(* Logix 5000 project; controller LeakTestAuto vendor 1 type 14 code 226 rev 37.11; software revision 37.01; part 4 of 13 *)

        [2].Detailed.element_data[13].result_measurement := 0.00085681677, [2].Detailed.element_data[14].Variable_code := 218, [2].Detailed.element_data[14].prec_code := 3, [2].Detailed.element_data[14].Unit_code := 41, [2].Detailed.element_data[14].result_measurement := 0.01094304, [2].Detailed.element_data[15].Variable_code := 295, [2].Detailed.element_data[15].prec_code := 3, [2].Detailed.element_data[15].Unit_code := 12, [2].Detailed.element_data[15].result_measurement := 5.073389, [3].UID := 10574, [3].Basic.unique_id := 10574, [3].Basic.channel_num := 1, [3].Basic.program_num := 2, [3].Basic.evaluation_code := 1, [3].Basic.test_port := 1, [3].Basic.year := 26, [3].Basic.month := 9, [3].Basic.date := 25, [3].Basic.hour := 12, [3].Basic.minute := 22, [3].Basic.second := 21, [3].Basic.flags := 12, [3].Basic.Num_tests := 1, [3].Basic.test_elements.test_type := 66, [3].Basic.test_elements.test_eval := 1, [3].Basic.test_elements.num_elements := 16, [3].Detailed.unique_id := 10574, [3].Detailed.num_elements := 16, [3].Detailed.Test_Type := 66, [3].Detailed.element_data[0].Variable_code := 61, [3].Detailed.element_data[0].prec_code := 2, [3].Detailed.element_data[0].Unit_code := 60, [3].Detailed.element_data[0].result_measurement := 0.11958182, [3].Detailed.element_data[1].Variable_code := 28, [3].Detailed.element_data[1].prec_code := 3, [3].Detailed.element_data[1].Unit_code := 41, [3].Detailed.element_data[1].result_measurement := 0.0037439167, [3].Detailed.element_data[2].Variable_code := 13, [3].Detailed.element_data[2].prec_code := 3, [3].Detailed.element_data[2].Unit_code := 12, [3].Detailed.element_data[2].result_measurement := 5.0675263, [3].Detailed.element_data[3].Variable_code := 75, [3].Detailed.element_data[3].prec_code := 2, [3].Detailed.element_data[3].Unit_code := 60, [3].Detailed.element_data[4].Variable_code := 60, [3].Detailed.element_data[4].prec_code := 2, [3].Detailed.element_data[4].Unit_code := 60, [3].Detailed.element_data[4].result_measurement := 0.1301989, [3].Detailed.element_data[5].Variable_code := 56, [3].Detailed.element_data[5].prec_code := 3, [3].Detailed.element_data[5].Unit_code := 41, [3].Detailed.element_data[5].result_measurement := 0.0020628795, [3].Detailed.element_data[6].Variable_code := 55, [3].Detailed.element_data[6].prec_code := 3, [3].Detailed.element_data[6].Unit_code := 12, [3].Detailed.element_data[6].result_measurement := 5.0675263, [3].Detailed.element_data[7].Variable_code := 58, [3].Detailed.element_data[7].prec_code := 2, [3].Detailed.element_data[7].Unit_code := 60, [3].Detailed.element_data[7].result_measurement := -1.0002404,
        [3].Detailed.element_data[8].Variable_code := 59, [3].Detailed.element_data[8].prec_code := 2, [3].Detailed.element_data[8].Unit_code := 60, [3].Detailed.element_data[8].result_measurement := 1.0002404, [3].Detailed.element_data[9].Variable_code := 12, [3].Detailed.element_data[9].prec_code := 3, [3].Detailed.element_data[9].Unit_code := 12, [3].Detailed.element_data[9].result_measurement := 5.000001, [3].Detailed.element_data[10].Variable_code := 62, [3].Detailed.element_data[10].prec_code := 2, [3].Detailed.element_data[10].Unit_code := 60, [3].Detailed.element_data[10].result_measurement := 1.0902061, [3].Detailed.element_data[11].Variable_code := 21, [3].Detailed.element_data[11].prec_code := 3, [3].Detailed.element_data[11].Unit_code := 41, [3].Detailed.element_data[11].result_measurement := 0.0015180558, [3].Detailed.element_data[12].Variable_code := 25, [3].Detailed.element_data[12].prec_code := 3, [3].Detailed.element_data[12].Unit_code := 41, [3].Detailed.element_data[12].result_measurement := 0.021727756, [3].Detailed.element_data[13].Variable_code := 216, [3].Detailed.element_data[13].prec_code := 3, [3].Detailed.element_data[13].Unit_code := 41, [3].Detailed.element_data[13].result_measurement := 0.00085681677, [3].Detailed.element_data[14].Variable_code := 218, [3].Detailed.element_data[14].prec_code := 3, [3].Detailed.element_data[14].Unit_code := 41, [3].Detailed.element_data[14].result_measurement := 0.01094304, [3].Detailed.element_data[15].Variable_code := 295, [3].Detailed.element_data[15].prec_code := 3, [3].Detailed.element_data[15].Unit_code := 12, [3].Detailed.element_data[15].result_measurement := 5.0734262, [4].UID := 10577, [4].Basic.unique_id := 10577, [4].Basic.channel_num := 1, [4].Basic.program_num := 2, [4].Basic.evaluation_code := 1, [4].Basic.test_port := 1, [4].Basic.year := 26, [4].Basic.month := 9, [4].Basic.date := 25, [4].Basic.hour := 12, [4].Basic.minute := 22, [4].Basic.second := 54, [4].Basic.flags := 12, [4].Basic.Num_tests := 1, [4].Basic.test_elements.test_type := 66, [4].Basic.test_elements.test_eval := 1, [4].Basic.test_elements.num_elements := 16, [4].Detailed.unique_id := 10577, [4].Detailed.num_elements := 16, [4].Detailed.Test_Type := 66, [4].Detailed.element_data[0].Variable_code := 61, [4].Detailed.element_data[0].prec_code := 2, [4].Detailed.element_data[0].Unit_code := 60, [4].Detailed.element_data[0].result_measurement := 0.10728836, [4].Detailed.element_data[1].Variable_code := 28, [4].Detailed.element_data[1].prec_code := 3, [4].Detailed.element_data[1].Unit_code := 41, [4].Detailed.element_data[1].result_measurement := 0.0035157427,
        [4].Detailed.element_data[2].Variable_code := 13, [4].Detailed.element_data[2].prec_code := 3, [4].Detailed.element_data[2].Unit_code := 12, [4].Detailed.element_data[2].result_measurement := 5.0673585, [4].Detailed.element_data[3].Variable_code := 75, [4].Detailed.element_data[3].prec_code := 2, [4].Detailed.element_data[3].Unit_code := 60, [4].Detailed.element_data[4].Variable_code := 60, [4].Detailed.element_data[4].prec_code := 2, [4].Detailed.element_data[4].Unit_code := 60, [4].Detailed.element_data[4].result_measurement := 0.093877316, [4].Detailed.element_data[5].Variable_code := 56, [4].Detailed.element_data[5].prec_code := 3, [4].Detailed.element_data[5].Unit_code := 41, [4].Detailed.element_data[5].result_measurement := 0.0017276034, [4].Detailed.element_data[6].Variable_code := 55, [4].Detailed.element_data[6].prec_code := 3, [4].Detailed.element_data[6].Unit_code := 12, [4].Detailed.element_data[6].result_measurement := 5.0673585, [4].Detailed.element_data[7].Variable_code := 58, [4].Detailed.element_data[7].prec_code := 2, [4].Detailed.element_data[7].Unit_code := 60, [4].Detailed.element_data[7].result_measurement := -1.0002404, [4].Detailed.element_data[8].Variable_code := 59, [4].Detailed.element_data[8].prec_code := 2, [4].Detailed.element_data[8].Unit_code := 60, [4].Detailed.element_data[8].result_measurement := 1.0002404, [4].Detailed.element_data[9].Variable_code := 12, [4].Detailed.element_data[9].prec_code := 3, [4].Detailed.element_data[9].Unit_code := 12, [4].Detailed.element_data[9].result_measurement := 5.000001, [4].Detailed.element_data[10].Variable_code := 62, [4].Detailed.element_data[10].prec_code := 2, [4].Detailed.element_data[10].Unit_code := 60, [4].Detailed.element_data[10].result_measurement := 1.0902061, [4].Detailed.element_data[11].Variable_code := 21, [4].Detailed.element_data[11].prec_code := 3, [4].Detailed.element_data[11].Unit_code := 41, [4].Detailed.element_data[11].result_measurement := 0.0015180558, [4].Detailed.element_data[12].Variable_code := 25, [4].Detailed.element_data[12].prec_code := 3, [4].Detailed.element_data[12].Unit_code := 41, [4].Detailed.element_data[12].result_measurement := 0.021727756, [4].Detailed.element_data[13].Variable_code := 216, [4].Detailed.element_data[13].prec_code := 3, [4].Detailed.element_data[13].Unit_code := 41, [4].Detailed.element_data[13].result_measurement := 0.00085681677, [4].Detailed.element_data[14].Variable_code := 218, [4].Detailed.element_data[14].prec_code := 3, [4].Detailed.element_data[14].Unit_code := 41, [4].Detailed.element_data[14].result_measurement := 0.01094304, [4].Detailed.element_data[15].Variable_code := 295, [4].Detailed.element_data[15].prec_code := 3, [4].Detailed.element_data[15].Unit_code := 12, [4].Detailed.element_data[15].result_measurement := 5.073468, [5].UID := 10580, [5].Basic.unique_id := 10580, [5].Basic.channel_num := 1, [5].Basic.program_num := 2, [5].Basic.evaluation_code := 1,
        [5].Basic.test_port := 1, [5].Basic.year := 26, [5].Basic.month := 9, [5].Basic.date := 25, [5].Basic.hour := 12, [5].Basic.minute := 27, [5].Basic.second := 36, [5].Basic.flags := 12, [5].Basic.Num_tests := 1, [5].Basic.test_elements.test_type := 66, [5].Basic.test_elements.test_eval := 1, [5].Basic.test_elements.num_elements := 16, [5].Detailed.unique_id := 10580, [5].Detailed.num_elements := 16, [5].Detailed.Test_Type := 66, [5].Detailed.element_data[0].Variable_code := 61, [5].Detailed.element_data[0].prec_code := 2, [5].Detailed.element_data[0].Unit_code := 60, [5].Detailed.element_data[0].result_measurement := 0.10281801, [5].Detailed.element_data[1].Variable_code := 28, [5].Detailed.element_data[1].prec_code := 3, [5].Detailed.element_data[1].Unit_code := 41, [5].Detailed.element_data[1].result_measurement := 0.003427267, [5].Detailed.element_data[2].Variable_code := 13, [5].Detailed.element_data[2].prec_code := 3, [5].Detailed.element_data[2].Unit_code := 12, [5].Detailed.element_data[2].result_measurement := 5.064076, [5].Detailed.element_data[3].Variable_code := 75, [5].Detailed.element_data[3].prec_code := 2, [5].Detailed.element_data[3].Unit_code := 60, [5].Detailed.element_data[4].Variable_code := 60, [5].Detailed.element_data[4].prec_code := 2, [5].Detailed.element_data[4].Unit_code := 60, [5].Detailed.element_data[4].result_measurement := 0.08773059, [5].Detailed.element_data[5].Variable_code := 56, [5].Detailed.element_data[5].prec_code := 3, [5].Detailed.element_data[5].Unit_code := 41, [5].Detailed.element_data[5].result_measurement := 0.001671724, [5].Detailed.element_data[6].Variable_code := 55, [5].Detailed.element_data[6].prec_code := 3, [5].Detailed.element_data[6].Unit_code := 12, [5].Detailed.element_data[6].result_measurement := 5.064076, [5].Detailed.element_data[7].Variable_code := 58, [5].Detailed.element_data[7].prec_code := 2, [5].Detailed.element_data[7].Unit_code := 60, [5].Detailed.element_data[7].result_measurement := -1.0002404, [5].Detailed.element_data[8].Variable_code := 59, [5].Detailed.element_data[8].prec_code := 2, [5].Detailed.element_data[8].Unit_code := 60, [5].Detailed.element_data[8].result_measurement := 1.0002404, [5].Detailed.element_data[9].Variable_code := 12, [5].Detailed.element_data[9].prec_code := 3, [5].Detailed.element_data[9].Unit_code := 12, [5].Detailed.element_data[9].result_measurement := 5.000001, [5].Detailed.element_data[10].Variable_code := 62, [5].Detailed.element_data[10].prec_code := 2, [5].Detailed.element_data[10].Unit_code := 60, [5].Detailed.element_data[10].result_measurement := 1.0902061, [5].Detailed.element_data[11].Variable_code := 21, [5].Detailed.element_data[11].prec_code := 3,
        [5].Detailed.element_data[11].Unit_code := 41, [5].Detailed.element_data[11].result_measurement := 0.0015180558, [5].Detailed.element_data[12].Variable_code := 25, [5].Detailed.element_data[12].prec_code := 3, [5].Detailed.element_data[12].Unit_code := 41, [5].Detailed.element_data[12].result_measurement := 0.021727756, [5].Detailed.element_data[13].Variable_code := 216, [5].Detailed.element_data[13].prec_code := 3, [5].Detailed.element_data[13].Unit_code := 41, [5].Detailed.element_data[13].result_measurement := 0.00085681677, [5].Detailed.element_data[14].Variable_code := 218, [5].Detailed.element_data[14].prec_code := 3, [5].Detailed.element_data[14].Unit_code := 41, [5].Detailed.element_data[14].result_measurement := 0.01094304, [5].Detailed.element_data[15].Variable_code := 295, [5].Detailed.element_data[15].prec_code := 3, [5].Detailed.element_data[15].Unit_code := 12, [5].Detailed.element_data[15].result_measurement := 5.0706367, [6].UID := 10583, [6].Basic.unique_id := 10583, [6].Basic.channel_num := 1, [6].Basic.program_num := 2, [6].Basic.evaluation_code := 1, [6].Basic.test_port := 1, [6].Basic.year := 26, [6].Basic.month := 9, [6].Basic.date := 25, [6].Basic.hour := 12, [6].Basic.minute := 28, [6].Basic.second := 6, [6].Basic.flags := 12, [6].Basic.Num_tests := 1, [6].Basic.test_elements.test_type := 66, [6].Basic.test_elements.test_eval := 1, [6].Basic.test_elements.num_elements := 16, [6].Detailed.unique_id := 10583, [6].Detailed.num_elements := 16, [6].Detailed.Test_Type := 66, [6].Detailed.element_data[0].Variable_code := 61, [6].Detailed.element_data[0].prec_code := 2, [6].Detailed.element_data[0].Unit_code := 60, [6].Detailed.element_data[0].result_measurement := 0.11622906, [6].Detailed.element_data[1].Variable_code := 28, [6].Detailed.element_data[1].prec_code := 3, [6].Detailed.element_data[1].Unit_code := 41, [6].Detailed.element_data[1].result_measurement := 0.0036740676, [6].Detailed.element_data[2].Variable_code := 13, [6].Detailed.element_data[2].prec_code := 3, [6].Detailed.element_data[2].Unit_code := 12, [6].Detailed.element_data[2].result_measurement := 5.0649743, [6].Detailed.element_data[3].Variable_code := 75, [6].Detailed.element_data[3].prec_code := 2, [6].Detailed.element_data[3].Unit_code := 60, [6].Detailed.element_data[4].Variable_code := 60, [6].Detailed.element_data[4].prec_code := 2, [6].Detailed.element_data[4].Unit_code := 60, [6].Detailed.element_data[4].result_measurement := 0.10114163, [6].Detailed.element_data[5].Variable_code := 56, [6].Detailed.element_data[5].prec_code := 3, [6].Detailed.element_data[5].Unit_code := 41,
        [6].Detailed.element_data[5].result_measurement := 0.001792796, [6].Detailed.element_data[6].Variable_code := 55, [6].Detailed.element_data[6].prec_code := 3, [6].Detailed.element_data[6].Unit_code := 12, [6].Detailed.element_data[6].result_measurement := 5.0649743, [6].Detailed.element_data[7].Variable_code := 58, [6].Detailed.element_data[7].prec_code := 2, [6].Detailed.element_data[7].Unit_code := 60, [6].Detailed.element_data[7].result_measurement := -1.0002404, [6].Detailed.element_data[8].Variable_code := 59, [6].Detailed.element_data[8].prec_code := 2, [6].Detailed.element_data[8].Unit_code := 60, [6].Detailed.element_data[8].result_measurement := 1.0002404, [6].Detailed.element_data[9].Variable_code := 12, [6].Detailed.element_data[9].prec_code := 3, [6].Detailed.element_data[9].Unit_code := 12, [6].Detailed.element_data[9].result_measurement := 5.000001, [6].Detailed.element_data[10].Variable_code := 62, [6].Detailed.element_data[10].prec_code := 2, [6].Detailed.element_data[10].Unit_code := 60, [6].Detailed.element_data[10].result_measurement := 1.0902061, [6].Detailed.element_data[11].Variable_code := 21, [6].Detailed.element_data[11].prec_code := 3, [6].Detailed.element_data[11].Unit_code := 41, [6].Detailed.element_data[11].result_measurement := 0.0015180558, [6].Detailed.element_data[12].Variable_code := 25, [6].Detailed.element_data[12].prec_code := 3, [6].Detailed.element_data[12].Unit_code := 41, [6].Detailed.element_data[12].result_measurement := 0.021727756, [6].Detailed.element_data[13].Variable_code := 216, [6].Detailed.element_data[13].prec_code := 3, [6].Detailed.element_data[13].Unit_code := 41, [6].Detailed.element_data[13].result_measurement := 0.00085681677, [6].Detailed.element_data[14].Variable_code := 218, [6].Detailed.element_data[14].prec_code := 3, [6].Detailed.element_data[14].Unit_code := 41, [6].Detailed.element_data[14].result_measurement := 0.01094304, [6].Detailed.element_data[15].Variable_code := 295, [6].Detailed.element_data[15].prec_code := 3, [6].Detailed.element_data[15].Unit_code := 12, [6].Detailed.element_data[15].result_measurement := 5.0712004, [7].UID := 10586, [7].Basic.unique_id := 10586, [7].Basic.channel_num := 1, [7].Basic.program_num := 2, [7].Basic.evaluation_code := 1, [7].Basic.test_port := 1, [7].Basic.year := 26, [7].Basic.month := 9, [7].Basic.date := 25, [7].Basic.hour := 12, [7].Basic.minute := 38, [7].Basic.second := 12, [7].Basic.flags := 12, [7].Basic.Num_tests := 1, [7].Basic.test_elements.test_type := 66, [7].Basic.test_elements.test_eval := 1, [7].Basic.test_elements.num_elements := 16, [7].Detailed.unique_id := 10586, [7].Detailed.num_elements := 16,
        [7].Detailed.Test_Type := 66, [7].Detailed.element_data[0].Variable_code := 61, [7].Detailed.element_data[0].prec_code := 2, [7].Detailed.element_data[0].Unit_code := 60, [7].Detailed.element_data[0].result_measurement := 0.11678785, [7].Detailed.element_data[1].Variable_code := 28, [7].Detailed.element_data[1].prec_code := 3, [7].Detailed.element_data[1].Unit_code := 41, [7].Detailed.element_data[1].result_measurement := 0.0036833808, [7].Detailed.element_data[2].Variable_code := 13, [7].Detailed.element_data[2].prec_code := 3, [7].Detailed.element_data[2].Unit_code := 12, [7].Detailed.element_data[2].result_measurement := 5.063303, [7].Detailed.element_data[3].Variable_code := 75, [7].Detailed.element_data[3].prec_code := 2, [7].Detailed.element_data[3].Unit_code := 60, [7].Detailed.element_data[4].Variable_code := 60, [7].Detailed.element_data[4].prec_code := 2, [7].Detailed.element_data[4].Unit_code := 60, [7].Detailed.element_data[4].result_measurement := 0.10617077, [7].Detailed.element_data[5].Variable_code := 56, [7].Detailed.element_data[5].prec_code := 3, [7].Detailed.element_data[5].Unit_code := 41, [7].Detailed.element_data[5].result_measurement := 0.0018440187, [7].Detailed.element_data[6].Variable_code := 55, [7].Detailed.element_data[6].prec_code := 3, [7].Detailed.element_data[6].Unit_code := 12, [7].Detailed.element_data[6].result_measurement := 5.063303, [7].Detailed.element_data[7].Variable_code := 58, [7].Detailed.element_data[7].prec_code := 2, [7].Detailed.element_data[7].Unit_code := 60, [7].Detailed.element_data[7].result_measurement := -1.0002404, [7].Detailed.element_data[8].Variable_code := 59, [7].Detailed.element_data[8].prec_code := 2, [7].Detailed.element_data[8].Unit_code := 60, [7].Detailed.element_data[8].result_measurement := 1.0002404, [7].Detailed.element_data[9].Variable_code := 12, [7].Detailed.element_data[9].prec_code := 3, [7].Detailed.element_data[9].Unit_code := 12, [7].Detailed.element_data[9].result_measurement := 5.000001, [7].Detailed.element_data[10].Variable_code := 62, [7].Detailed.element_data[10].prec_code := 2, [7].Detailed.element_data[10].Unit_code := 60, [7].Detailed.element_data[10].result_measurement := 1.0902061, [7].Detailed.element_data[11].Variable_code := 21, [7].Detailed.element_data[11].prec_code := 3, [7].Detailed.element_data[11].Unit_code := 41, [7].Detailed.element_data[11].result_measurement := 0.0015180558, [7].Detailed.element_data[12].Variable_code := 25, [7].Detailed.element_data[12].prec_code := 3, [7].Detailed.element_data[12].Unit_code := 41, [7].Detailed.element_data[12].result_measurement := 0.021727756, [7].Detailed.element_data[13].Variable_code := 216, [7].Detailed.element_data[13].prec_code := 3, [7].Detailed.element_data[13].Unit_code := 41, [7].Detailed.element_data[13].result_measurement := 0.00085681677, [7].Detailed.element_data[14].Variable_code := 218, [7].Detailed.element_data[14].prec_code := 3, [7].Detailed.element_data[14].Unit_code := 41, [7].Detailed.element_data[14].result_measurement := 0.01094304,
        [7].Detailed.element_data[15].Variable_code := 295, [7].Detailed.element_data[15].prec_code := 3, [7].Detailed.element_data[15].Unit_code := 12, [7].Detailed.element_data[15].result_measurement := 5.0700407, [8].UID := 10589, [8].Basic.unique_id := 10589, [8].Basic.channel_num := 1, [8].Basic.program_num := 2, [8].Basic.evaluation_code := 1, [8].Basic.test_port := 1, [8].Basic.year := 26, [8].Basic.month := 9, [8].Basic.date := 25, [8].Basic.hour := 12, [8].Basic.minute := 39, [8].Basic.second := 1, [8].Basic.flags := 12, [8].Basic.Num_tests := 1, [8].Basic.test_elements.test_type := 66, [8].Basic.test_elements.test_eval := 1, [8].Basic.test_elements.num_elements := 16, [8].Detailed.unique_id := 10589, [8].Detailed.num_elements := 16, [8].Detailed.Test_Type := 66, [8].Detailed.element_data[0].Variable_code := 61, [8].Detailed.element_data[0].prec_code := 2, [8].Detailed.element_data[0].Unit_code := 60, [8].Detailed.element_data[0].result_measurement := 0.11175871, [8].Detailed.element_data[1].Variable_code := 28, [8].Detailed.element_data[1].prec_code := 3, [8].Detailed.element_data[1].Unit_code := 41, [8].Detailed.element_data[1].result_measurement := 0.0035949051, [8].Detailed.element_data[2].Variable_code := 13, [8].Detailed.element_data[2].prec_code := 3, [8].Detailed.element_data[2].Unit_code := 12, [8].Detailed.element_data[2].result_measurement := 5.0623946, [8].Detailed.element_data[3].Variable_code := 75, [8].Detailed.element_data[3].prec_code := 2, [8].Detailed.element_data[3].Unit_code := 60, [8].Detailed.element_data[4].Variable_code := 60, [8].Detailed.element_data[4].prec_code := 2, [8].Detailed.element_data[4].Unit_code := 60, [8].Detailed.element_data[4].result_measurement := 0.11175871, [8].Detailed.element_data[5].Variable_code := 56, [8].Detailed.element_data[5].prec_code := 3, [8].Detailed.element_data[5].Unit_code := 41, [8].Detailed.element_data[5].result_measurement := 0.0018952414, [8].Detailed.element_data[6].Variable_code := 55, [8].Detailed.element_data[6].prec_code := 3, [8].Detailed.element_data[6].Unit_code := 12, [8].Detailed.element_data[6].result_measurement := 5.0623946, [8].Detailed.element_data[7].Variable_code := 58, [8].Detailed.element_data[7].prec_code := 2, [8].Detailed.element_data[7].Unit_code := 60, [8].Detailed.element_data[7].result_measurement := -1.0002404, [8].Detailed.element_data[8].Variable_code := 59, [8].Detailed.element_data[8].prec_code := 2, [8].Detailed.element_data[8].Unit_code := 60, [8].Detailed.element_data[8].result_measurement := 1.0002404, [8].Detailed.element_data[9].Variable_code := 12,
        [8].Detailed.element_data[9].prec_code := 3, [8].Detailed.element_data[9].Unit_code := 12, [8].Detailed.element_data[9].result_measurement := 5.000001, [8].Detailed.element_data[10].Variable_code := 62, [8].Detailed.element_data[10].prec_code := 2, [8].Detailed.element_data[10].Unit_code := 60, [8].Detailed.element_data[10].result_measurement := 1.0902061, [8].Detailed.element_data[11].Variable_code := 21, [8].Detailed.element_data[11].prec_code := 3, [8].Detailed.element_data[11].Unit_code := 41, [8].Detailed.element_data[11].result_measurement := 0.0015180558, [8].Detailed.element_data[12].Variable_code := 25, [8].Detailed.element_data[12].prec_code := 3, [8].Detailed.element_data[12].Unit_code := 41, [8].Detailed.element_data[12].result_measurement := 0.021727756, [8].Detailed.element_data[13].Variable_code := 216, [8].Detailed.element_data[13].prec_code := 3, [8].Detailed.element_data[13].Unit_code := 41, [8].Detailed.element_data[13].result_measurement := 0.00085681677, [8].Detailed.element_data[14].Variable_code := 218, [8].Detailed.element_data[14].prec_code := 3, [8].Detailed.element_data[14].Unit_code := 41, [8].Detailed.element_data[14].result_measurement := 0.01094304, [8].Detailed.element_data[15].Variable_code := 295, [8].Detailed.element_data[15].prec_code := 3, [8].Detailed.element_data[15].Unit_code := 12, [8].Detailed.element_data[15].result_measurement := 5.068914, [9].UID := 10592, [9].Basic.unique_id := 10592, [9].Basic.channel_num := 1, [9].Basic.program_num := 2, [9].Basic.evaluation_code := 1, [9].Basic.test_port := 1, [9].Basic.year := 26, [9].Basic.month := 9, [9].Basic.date := 25, [9].Basic.hour := 12, [9].Basic.minute := 39, [9].Basic.second := 32, [9].Basic.flags := 12, [9].Basic.Num_tests := 1, [9].Basic.test_elements.test_type := 66, [9].Basic.test_elements.test_eval := 1, [9].Basic.test_elements.num_elements := 16, [9].Detailed.unique_id := 10592, [9].Detailed.num_elements := 16, [9].Detailed.Test_Type := 66, [9].Detailed.element_data[0].Variable_code := 61, [9].Detailed.element_data[0].prec_code := 2, [9].Detailed.element_data[0].Unit_code := 60, [9].Detailed.element_data[0].result_measurement := 0.10728836, [9].Detailed.element_data[1].Variable_code := 28, [9].Detailed.element_data[1].prec_code := 3, [9].Detailed.element_data[1].Unit_code := 41, [9].Detailed.element_data[1].result_measurement := 0.003511086, [9].Detailed.element_data[2].Variable_code := 13, [9].Detailed.element_data[2].prec_code := 3, [9].Detailed.element_data[2].Unit_code := 12, [9].Detailed.element_data[2].result_measurement := 5.0658684, [9].Detailed.element_data[3].Variable_code := 75,
        [9].Detailed.element_data[3].prec_code := 2, [9].Detailed.element_data[3].Unit_code := 60, [9].Detailed.element_data[4].Variable_code := 60, [9].Detailed.element_data[4].prec_code := 2, [9].Detailed.element_data[4].Unit_code := 60, [9].Detailed.element_data[4].result_measurement := 0.12684613, [9].Detailed.element_data[5].Variable_code := 56, [9].Detailed.element_data[5].prec_code := 3, [9].Detailed.element_data[5].Unit_code := 41, [9].Detailed.element_data[5].result_measurement := 0.0020349398, [9].Detailed.element_data[6].Variable_code := 55, [9].Detailed.element_data[6].prec_code := 3, [9].Detailed.element_data[6].Unit_code := 12, [9].Detailed.element_data[6].result_measurement := 5.0658684, [9].Detailed.element_data[7].Variable_code := 58, [9].Detailed.element_data[7].prec_code := 2, [9].Detailed.element_data[7].Unit_code := 60, [9].Detailed.element_data[7].result_measurement := -1.0002404, [9].Detailed.element_data[8].Variable_code := 59, [9].Detailed.element_data[8].prec_code := 2, [9].Detailed.element_data[8].Unit_code := 60, [9].Detailed.element_data[8].result_measurement := 1.0002404, [9].Detailed.element_data[9].Variable_code := 12, [9].Detailed.element_data[9].prec_code := 3, [9].Detailed.element_data[9].Unit_code := 12, [9].Detailed.element_data[9].result_measurement := 5.000001, [9].Detailed.element_data[10].Variable_code := 62, [9].Detailed.element_data[10].prec_code := 2, [9].Detailed.element_data[10].Unit_code := 60, [9].Detailed.element_data[10].result_measurement := 1.0902061, [9].Detailed.element_data[11].Variable_code := 21, [9].Detailed.element_data[11].prec_code := 3, [9].Detailed.element_data[11].Unit_code := 41, [9].Detailed.element_data[11].result_measurement := 0.0015180558, [9].Detailed.element_data[12].Variable_code := 25, [9].Detailed.element_data[12].prec_code := 3, [9].Detailed.element_data[12].Unit_code := 41, [9].Detailed.element_data[12].result_measurement := 0.021727756, [9].Detailed.element_data[13].Variable_code := 216, [9].Detailed.element_data[13].prec_code := 3, [9].Detailed.element_data[13].Unit_code := 41, [9].Detailed.element_data[13].result_measurement := 0.00085681677, [9].Detailed.element_data[14].Variable_code := 218, [9].Detailed.element_data[14].prec_code := 3, [9].Detailed.element_data[14].Unit_code := 41, [9].Detailed.element_data[14].result_measurement := 0.01094304, [9].Detailed.element_data[15].Variable_code := 295, [9].Detailed.element_data[15].prec_code := 3, [9].Detailed.element_data[15].Unit_code := 12, [9].Detailed.element_data[15].result_measurement := 5.0730352);
   CTS2_ResultHistoryVol : udt_CTS_RESULT[10] := ([0].UID := 10564, [0].Basic.unique_id := 10564, [0].Basic.channel_num := 1, [0].Basic.program_num := 1, [0].Basic.evaluation_code := 1, [0].Basic.test_port := 1, [0].Basic.year := 26, [0].Basic.month := 9, [0].Basic.date := 25, [0].Basic.hour := 12, [0].Basic.minute := 21, [0].Basic.second := 12, [0].Basic.flags := 12, [0].Basic.Num_tests := 1, [0].Basic.test_elements.test_type := 69, [0].Basic.test_elements.test_eval := 1, [0].Basic.test_elements.num_elements := 4, [0].Detailed.unique_id := 10564, [0].Detailed.num_elements := 4, [0].Detailed.Test_Type := 69, [0].Detailed.element_data[0].Variable_code := 245, [0].Detailed.element_data[0].prec_code := 2, [0].Detailed.element_data[0].Unit_code := 165, [0].Detailed.element_data[0].result_measurement := 156.89374, [0].Detailed.element_data[1].Variable_code := 13, [0].Detailed.element_data[1].prec_code := 3, [0].Detailed.element_data[1].Unit_code := 12, [0].Detailed.element_data[1].result_measurement := 1.962753, [0].Detailed.element_data[2].Variable_code := 247, [0].Detailed.element_data[2].prec_code := 3, [0].Detailed.element_data[2].Unit_code := 12, [0].Detailed.element_data[2].result_measurement := 5.0421896, [0].Detailed.element_data[3].Variable_code := 295, [0].Detailed.element_data[3].prec_code := 3, [0].Detailed.element_data[3].Unit_code := 12, [0].Detailed.element_data[3].result_measurement := 5.0442944, [1].UID := 10567, [1].Basic.unique_id := 10567, [1].Basic.channel_num := 1, [1].Basic.program_num := 1, [1].Basic.evaluation_code := 1, [1].Basic.test_port := 1, [1].Basic.year := 26, [1].Basic.month := 9, [1].Basic.date := 25, [1].Basic.hour := 12, [1].Basic.minute := 21, [1].Basic.second := 33, [1].Basic.flags := 12, [1].Basic.Num_tests := 1, [1].Basic.test_elements.test_type := 69, [1].Basic.test_elements.test_eval := 1, [1].Basic.test_elements.num_elements := 4, [1].Detailed.unique_id := 10567, [1].Detailed.num_elements := 4, [1].Detailed.Test_Type := 69, [1].Detailed.element_data[0].Variable_code := 245, [1].Detailed.element_data[0].prec_code := 2, [1].Detailed.element_data[0].Unit_code := 165, [1].Detailed.element_data[0].result_measurement := 156.82765,
        [1].Detailed.element_data[1].Variable_code := 13, [1].Detailed.element_data[1].prec_code := 3, [1].Detailed.element_data[1].Unit_code := 12, [1].Detailed.element_data[1].result_measurement := 1.9633397, [1].Detailed.element_data[2].Variable_code := 247, [1].Detailed.element_data[2].prec_code := 3, [1].Detailed.element_data[2].Unit_code := 12, [1].Detailed.element_data[2].result_measurement := 5.0423994, [1].Detailed.element_data[3].Variable_code := 295, [1].Detailed.element_data[3].prec_code := 3, [1].Detailed.element_data[3].Unit_code := 12, [1].Detailed.element_data[3].result_measurement := 5.04469, [2].UID := 10570, [2].Basic.unique_id := 10570, [2].Basic.channel_num := 1, [2].Basic.program_num := 1, [2].Basic.evaluation_code := 1, [2].Basic.test_port := 1, [2].Basic.year := 26, [2].Basic.month := 9, [2].Basic.date := 25, [2].Basic.hour := 12, [2].Basic.minute := 21, [2].Basic.second := 54, [2].Basic.flags := 12, [2].Basic.Num_tests := 1, [2].Basic.test_elements.test_type := 69, [2].Basic.test_elements.test_eval := 1, [2].Basic.test_elements.num_elements := 4, [2].Detailed.unique_id := 10570, [2].Detailed.num_elements := 4, [2].Detailed.Test_Type := 69, [2].Detailed.element_data[0].Variable_code := 245, [2].Detailed.element_data[0].prec_code := 2, [2].Detailed.element_data[0].Unit_code := 165, [2].Detailed.element_data[0].result_measurement := 156.6537, [2].Detailed.element_data[1].Variable_code := 13, [2].Detailed.element_data[1].prec_code := 3, [2].Detailed.element_data[1].Unit_code := 12, [2].Detailed.element_data[1].result_measurement := 1.9648718, [2].Detailed.element_data[2].Variable_code := 247, [2].Detailed.element_data[2].prec_code := 3, [2].Detailed.element_data[2].Unit_code := 12, [2].Detailed.element_data[2].result_measurement := 5.0429163, [2].Detailed.element_data[3].Variable_code := 295, [2].Detailed.element_data[3].prec_code := 3, [2].Detailed.element_data[3].Unit_code := 12, [2].Detailed.element_data[3].result_measurement := 5.044765, [3].UID := 10573, [3].Basic.unique_id := 10573, [3].Basic.channel_num := 1, [3].Basic.program_num := 1, [3].Basic.evaluation_code := 1, [3].Basic.test_port := 1, [3].Basic.year := 26, [3].Basic.month := 9, [3].Basic.date := 25, [3].Basic.hour := 12, [3].Basic.minute := 22, [3].Basic.second := 15,
        [3].Basic.flags := 12, [3].Basic.Num_tests := 1, [3].Basic.test_elements.test_type := 69, [3].Basic.test_elements.test_eval := 1, [3].Basic.test_elements.num_elements := 4, [3].Detailed.unique_id := 10573, [3].Detailed.num_elements := 4, [3].Detailed.Test_Type := 69, [3].Detailed.element_data[0].Variable_code := 245, [3].Detailed.element_data[0].prec_code := 2, [3].Detailed.element_data[0].Unit_code := 165, [3].Detailed.element_data[0].result_measurement := 156.76877, [3].Detailed.element_data[1].Variable_code := 13, [3].Detailed.element_data[1].prec_code := 3, [3].Detailed.element_data[1].Unit_code := 12, [3].Detailed.element_data[1].result_measurement := 1.9644899, [3].Detailed.element_data[2].Variable_code := 247, [3].Detailed.element_data[2].prec_code := 3, [3].Detailed.element_data[2].Unit_code := 12, [3].Detailed.element_data[2].result_measurement := 5.0441966, [3].Detailed.element_data[3].Variable_code := 295, [3].Detailed.element_data[3].prec_code := 3, [3].Detailed.element_data[3].Unit_code := 12, [3].Detailed.element_data[3].result_measurement := 5.0450954, [4].UID := 10576, [4].Basic.unique_id := 10576, [4].Basic.channel_num := 1, [4].Basic.program_num := 1, [4].Basic.evaluation_code := 1, [4].Basic.test_port := 1, [4].Basic.year := 26, [4].Basic.month := 9, [4].Basic.date := 25, [4].Basic.hour := 12, [4].Basic.minute := 22, [4].Basic.second := 47, [4].Basic.flags := 12, [4].Basic.Num_tests := 1, [4].Basic.test_elements.test_type := 69, [4].Basic.test_elements.test_eval := 1, [4].Basic.test_elements.num_elements := 4, [4].Detailed.unique_id := 10576, [4].Detailed.num_elements := 4, [4].Detailed.Test_Type := 69, [4].Detailed.element_data[0].Variable_code := 245, [4].Detailed.element_data[0].prec_code := 2, [4].Detailed.element_data[0].Unit_code := 165, [4].Detailed.element_data[0].result_measurement := 154.13881, [4].Detailed.element_data[1].Variable_code := 13, [4].Detailed.element_data[1].prec_code := 3, [4].Detailed.element_data[1].Unit_code := 12, [4].Detailed.element_data[1].result_measurement := 1.9848579, [4].Detailed.element_data[2].Variable_code := 247, [4].Detailed.element_data[2].prec_code := 3, [4].Detailed.element_data[2].Unit_code := 12, [4].Detailed.element_data[2].result_measurement := 5.0442944, [4].Detailed.element_data[3].Variable_code := 295, [4].Detailed.element_data[3].prec_code := 3, [4].Detailed.element_data[3].Unit_code := 12, [4].Detailed.element_data[3].result_measurement := 5.0455236,
        [5].UID := 10579, [5].Basic.unique_id := 10579, [5].Basic.channel_num := 1, [5].Basic.program_num := 1, [5].Basic.evaluation_code := 1, [5].Basic.test_port := 1, [5].Basic.year := 26, [5].Basic.month := 9, [5].Basic.date := 25, [5].Basic.hour := 12, [5].Basic.minute := 27, [5].Basic.second := 29, [5].Basic.flags := 12, [5].Basic.Num_tests := 1, [5].Basic.test_elements.test_type := 69, [5].Basic.test_elements.test_eval := 1, [5].Basic.test_elements.num_elements := 4, [5].Detailed.unique_id := 10579, [5].Detailed.num_elements := 4, [5].Detailed.Test_Type := 69, [5].Detailed.element_data[0].Variable_code := 245, [5].Detailed.element_data[0].prec_code := 2, [5].Detailed.element_data[0].Unit_code := 165, [5].Detailed.element_data[0].result_measurement := 157.14537, [5].Detailed.element_data[1].Variable_code := 13, [5].Detailed.element_data[1].prec_code := 3, [5].Detailed.element_data[1].Unit_code := 12, [5].Detailed.element_data[1].result_measurement := 1.9622269, [5].Detailed.element_data[2].Variable_code := 247, [5].Detailed.element_data[2].prec_code := 3, [5].Detailed.element_data[2].Unit_code := 12, [5].Detailed.element_data[2].result_measurement := 5.0457754, [5].Detailed.element_data[3].Variable_code := 295, [5].Detailed.element_data[3].prec_code := 3, [5].Detailed.element_data[3].Unit_code := 12, [5].Detailed.element_data[3].result_measurement := 5.0467906, [6].UID := 10582, [6].Basic.unique_id := 10582, [6].Basic.channel_num := 1, [6].Basic.program_num := 1, [6].Basic.evaluation_code := 1, [6].Basic.test_port := 1, [6].Basic.year := 26, [6].Basic.month := 9, [6].Basic.date := 25, [6].Basic.hour := 12, [6].Basic.minute := 28, [6].Basic.flags := 12, [6].Basic.Num_tests := 1, [6].Basic.test_elements.test_type := 69, [6].Basic.test_elements.test_eval := 1, [6].Basic.test_elements.num_elements := 4, [6].Detailed.unique_id := 10582, [6].Detailed.num_elements := 4, [6].Detailed.Test_Type := 69, [6].Detailed.element_data[0].Variable_code := 245, [6].Detailed.element_data[0].prec_code := 2, [6].Detailed.element_data[0].Unit_code := 165, [6].Detailed.element_data[0].result_measurement := 156.1754, [6].Detailed.element_data[1].Variable_code := 13,
        [6].Detailed.element_data[1].prec_code := 3, [6].Detailed.element_data[1].Unit_code := 12, [6].Detailed.element_data[1].result_measurement := 1.9685458, [6].Detailed.element_data[2].Variable_code := 247, [6].Detailed.element_data[2].prec_code := 3, [6].Detailed.element_data[2].Unit_code := 12, [6].Detailed.element_data[2].result_measurement := 5.04293, [6].Detailed.element_data[3].Variable_code := 295, [6].Detailed.element_data[3].prec_code := 3, [6].Detailed.element_data[3].Unit_code := 12, [6].Detailed.element_data[3].result_measurement := 5.0441875, [7].UID := 10585, [7].Basic.unique_id := 10585, [7].Basic.channel_num := 1, [7].Basic.program_num := 1, [7].Basic.evaluation_code := 1, [7].Basic.test_port := 1, [7].Basic.year := 26, [7].Basic.month := 9, [7].Basic.date := 25, [7].Basic.hour := 12, [7].Basic.minute := 38, [7].Basic.second := 5, [7].Basic.flags := 12, [7].Basic.Num_tests := 1, [7].Basic.test_elements.test_type := 69, [7].Basic.test_elements.test_eval := 1, [7].Basic.test_elements.num_elements := 4, [7].Detailed.unique_id := 10585, [7].Detailed.num_elements := 4, [7].Detailed.Test_Type := 69, [7].Detailed.element_data[0].Variable_code := 245, [7].Detailed.element_data[0].prec_code := 2, [7].Detailed.element_data[0].Unit_code := 165, [7].Detailed.element_data[0].result_measurement := 156.68964, [7].Detailed.element_data[1].Variable_code := 13, [7].Detailed.element_data[1].prec_code := 3, [7].Detailed.element_data[1].Unit_code := 12, [7].Detailed.element_data[1].result_measurement := 1.9655237, [7].Detailed.element_data[2].Variable_code := 247, [7].Detailed.element_data[2].prec_code := 3, [7].Detailed.element_data[2].Unit_code := 12, [7].Detailed.element_data[2].result_measurement := 5.0452957, [7].Detailed.element_data[3].Variable_code := 295, [7].Detailed.element_data[3].prec_code := 3, [7].Detailed.element_data[3].Unit_code := 12, [7].Detailed.element_data[3].result_measurement := 5.046395, [8].UID := 10588, [8].Basic.unique_id := 10588, [8].Basic.channel_num := 1, [8].Basic.program_num := 1, [8].Basic.evaluation_code := 1, [8].Basic.test_port := 1, [8].Basic.year := 26, [8].Basic.month := 9, [8].Basic.date := 25, [8].Basic.hour := 12, [8].Basic.minute := 38, [8].Basic.second := 54, [8].Basic.flags := 12,
        [8].Basic.Num_tests := 1, [8].Basic.test_elements.test_type := 69, [8].Basic.test_elements.test_eval := 1, [8].Basic.test_elements.num_elements := 4, [8].Detailed.unique_id := 10588, [8].Detailed.num_elements := 4, [8].Detailed.Test_Type := 69, [8].Detailed.element_data[0].Variable_code := 245, [8].Detailed.element_data[0].prec_code := 2, [8].Detailed.element_data[0].Unit_code := 165, [8].Detailed.element_data[0].result_measurement := 156.9294, [8].Detailed.element_data[1].Variable_code := 13, [8].Detailed.element_data[1].prec_code := 3, [8].Detailed.element_data[1].Unit_code := 12, [8].Detailed.element_data[1].result_measurement := 1.9627343, [8].Detailed.element_data[2].Variable_code := 247, [8].Detailed.element_data[2].prec_code := 3, [8].Detailed.element_data[2].Unit_code := 12, [8].Detailed.element_data[2].result_measurement := 5.0428414, [8].Detailed.element_data[3].Variable_code := 295, [8].Detailed.element_data[3].prec_code := 3, [8].Detailed.element_data[3].Unit_code := 12, [8].Detailed.element_data[3].result_measurement := 5.0439687, [9].UID := 10591, [9].Basic.unique_id := 10591, [9].Basic.channel_num := 1, [9].Basic.program_num := 1, [9].Basic.evaluation_code := 1, [9].Basic.test_port := 1, [9].Basic.year := 26, [9].Basic.month := 9, [9].Basic.date := 25, [9].Basic.hour := 12, [9].Basic.minute := 39, [9].Basic.second := 25, [9].Basic.flags := 12, [9].Basic.Num_tests := 1, [9].Basic.test_elements.test_type := 69, [9].Basic.test_elements.test_eval := 1, [9].Basic.test_elements.num_elements := 4, [9].Detailed.unique_id := 10591, [9].Detailed.num_elements := 4, [9].Detailed.Test_Type := 69, [9].Detailed.element_data[0].Variable_code := 245, [9].Detailed.element_data[0].prec_code := 2, [9].Detailed.element_data[0].Unit_code := 165, [9].Detailed.element_data[0].result_measurement := 191.42384, [9].Detailed.element_data[1].Variable_code := 13, [9].Detailed.element_data[1].prec_code := 3, [9].Detailed.element_data[1].Unit_code := 12, [9].Detailed.element_data[1].result_measurement := 1.7302344, [9].Detailed.element_data[2].Variable_code := 247, [9].Detailed.element_data[2].prec_code := 3, [9].Detailed.element_data[2].Unit_code := 12, [9].Detailed.element_data[2].result_measurement := 5.0423155, [9].Detailed.element_data[3].Variable_code := 295, [9].Detailed.element_data[3].prec_code := 3, [9].Detailed.element_data[3].Unit_code := 12, [9].Detailed.element_data[3].result_measurement := 5.0434656);
   CTS2_Seq : udt_SequenceStructure_X64 := (CycleDone := 1, CurrentStep := 9000, NextStep := 9000, ONS := -32767, StepHistory[0] := 1000, StepHistory[1] := 1010, StepHistory[2] := 1020, StepHistory[3] := 1030, StepHistory[4] := 2000, StepHistory[5] := 2010, StepHistory[6] := 2020, StepHistory[7] := 2030, StepHistory[8] := 2000, StepHistory[9] := 2010, StepHistory[10] := 2020, StepHistory[11] := 2030, StepHistory[12] := 9000, StepHistory[13] := 1000, StepHistory[14] := 1010, StepHistory[15] := 1020, StepHistory[16] := 1030, StepHistory[17] := 2000, StepHistory[18] := 2010, StepHistory[19] := 2020, StepHistory[20] := 2030, StepHistory[21] := 2000, StepHistory[22] := 2010, StepHistory[23] := 2020, StepHistory[24] := 2030, StepHistory[25] := 9000, StepHistory[26] := 1000, StepHistory[27] := 1010, StepHistory[28] := 1020, StepHistory[29] := 1030, StepHistory[30] := 2000, StepHistory[31] := 2010, StepHistory[32] := 2020, StepHistory[33] := 2030, StepHistory[34] := 2000, StepHistory[35] := 2010, StepHistory[36] := 2020, StepHistory[37] := 2030, StepHistory[38] := 9000, StepHistory[39] := 1000, StepHistory[40] := 1010, StepHistory[41] := 1020, StepHistory[42] := 1030, StepHistory[43] := 2000, StepHistory[44] := 2010, StepHistory[45] := 2020, StepHistory[46] := 2030, StepHistory[47] := 2000, StepHistory[48] := 2010, StepHistory[49] := 2020, StepHistory[50] := 2030, StepHistory[51] := 9000, StepHistory[52] := 1000, StepHistory[53] := 1010, StepHistory[54] := 1020, StepHistory[55] := 1030,
        StepHistory[56] := 2000, StepHistory[57] := 2010, StepHistory[58] := 2020, StepHistory[59] := 2030, StepHistory[60] := 2000, StepHistory[61] := 2010, StepHistory[62] := 2020, StepHistory[63] := 2030, AverageCycleTime := 0.442, CycleTimeHistory[0] := 2.21, CycleTimeHistory[1] := 2.21, StepTimeHistory[1] := 0.2, StepTimeHistory[2] := 0.2, StepTimeHistory[3] := 0.2, StepTimeHistory[5] := 0.999, StepTimeHistory[6] := 0.999, StepTimeHistory[7] := 0.999, StepTimeHistory[9] := 0.999, StepTimeHistory[10] := 0.999, StepTimeHistory[11] := 0.999, StepTimeHistory[12] := 0.999, StepTimeHistory[14] := 0.199, StepTimeHistory[15] := 0.199, StepTimeHistory[16] := 0.199, StepTimeHistory[18] := 0.999, StepTimeHistory[19] := 0.999, StepTimeHistory[20] := 0.999, StepTimeHistory[22] := 0.999, StepTimeHistory[23] := 0.999, StepTimeHistory[24] := 0.999, StepTimeHistory[25] := 0.999, StepTimeHistory[27] := 0.199, StepTimeHistory[28] := 0.199, StepTimeHistory[29] := 0.199, StepTimeHistory[31] := 0.999, StepTimeHistory[32] := 0.999, StepTimeHistory[33] := 0.999, StepTimeHistory[35] := 0.999, StepTimeHistory[36] := 0.999, StepTimeHistory[37] := 0.999, StepTimeHistory[38] := 0.999, StepTimeHistory[40] := 0.199, StepTimeHistory[41] := 0.199, StepTimeHistory[42] := 0.199, StepTimeHistory[44] := 0.999, StepTimeHistory[45] := 0.999, StepTimeHistory[46] := 0.999, StepTimeHistory[48] := 1.0, StepTimeHistory[49] := 1.0, StepTimeHistory[50] := 1.0, StepTimeHistory[51] := 1.0, StepTimeHistory[53] := 0.199, StepTimeHistory[54] := 0.199, StepTimeHistory[55] := 0.199, StepTimeHistory[57] := 1.0, StepTimeHistory[58] := 1.0, StepTimeHistory[59] := 1.0, StepTimeHistory[61] := 0.999, StepTimeHistory[62] := 0.999, StepTimeHistory[63] := 0.999,
        StepTimer.PRE := 999999999, CycleTimer.PRE := 999999999);
   CTS2_SeqUID : DINT := 10590;
   CTS2_UIDMsg : MESSAGE;
        MessageParameters(ServiceCode := 16#0010, LocalElement := CTS2_Result.UID, ...)
   CTS2_WriteMsg : MESSAGE;
        MessageParameters(ServiceCode := 16#0010, LocalElement := CTS2_BarcodeWrite.DATA[0], ...)
   CTS_NoResult : udt_CTS_RESULT;
   CTS_ResultDump : udt_CTS_RESULT := (UID := 10562, Basic.unique_id := 10562, Basic.channel_num := 1, Basic.program_num := 2, Basic.evaluation_code := 2, Basic.test_port := 1, Basic.year := 26, Basic.month := 9, Basic.date := 25, Basic.hour := 12, Basic.minute := 20, Basic.second := 58, Basic.flags := 12, Basic.Num_tests := 1, Basic.test_elements.test_type := 66, Basic.test_elements.test_eval := 2, Basic.test_elements.num_elements := 16, Detailed.unique_id := 10562, Detailed.num_elements := 16, Detailed.Test_Type := 66, Detailed.element_data[0].Variable_code := 61, Detailed.element_data[0].prec_code := 2, Detailed.element_data[0].Unit_code := 60, Detailed.element_data[0].result_measurement := 4.5916066, Detailed.element_data[1].Variable_code := 28, Detailed.element_data[1].prec_code := 3, Detailed.element_data[1].Unit_code := 41, Detailed.element_data[1].result_measurement := 0.08663628, Detailed.element_data[2].Variable_code := 13, Detailed.element_data[2].prec_code := 3, Detailed.element_data[2].Unit_code := 12, Detailed.element_data[2].result_measurement := 4.954045, Detailed.element_data[3].Variable_code := 75, Detailed.element_data[3].prec_code := 2, Detailed.element_data[3].Unit_code := 60, Detailed.element_data[4].Variable_code := 60, Detailed.element_data[4].prec_code := 2, Detailed.element_data[4].Unit_code := 60, Detailed.element_data[4].result_measurement := 4.707277, Detailed.element_data[5].Variable_code := 56, Detailed.element_data[5].prec_code := 3, Detailed.element_data[5].Unit_code := 41, Detailed.element_data[5].result_measurement := 0.044410117, Detailed.element_data[6].Variable_code := 55, Detailed.element_data[6].prec_code := 3, Detailed.element_data[6].Unit_code := 12, Detailed.element_data[6].result_measurement := 4.954045, Detailed.element_data[7].Variable_code := 58, Detailed.element_data[7].prec_code := 2, Detailed.element_data[7].Unit_code := 60, Detailed.element_data[7].result_measurement := -1.0002404, Detailed.element_data[8].Variable_code := 59, Detailed.element_data[8].prec_code := 2, Detailed.element_data[8].Unit_code := 60, Detailed.element_data[8].result_measurement := 1.0002404, Detailed.element_data[9].Variable_code := 12, Detailed.element_data[9].prec_code := 3, Detailed.element_data[9].Unit_code := 12, Detailed.element_data[9].result_measurement := 5.000001, Detailed.element_data[10].Variable_code := 62,
        Detailed.element_data[10].prec_code := 2, Detailed.element_data[10].Unit_code := 60, Detailed.element_data[10].result_measurement := 1.0902061, Detailed.element_data[11].Variable_code := 21, Detailed.element_data[11].prec_code := 3, Detailed.element_data[11].Unit_code := 41, Detailed.element_data[11].result_measurement := 0.0015180558, Detailed.element_data[12].Variable_code := 25, Detailed.element_data[12].prec_code := 3, Detailed.element_data[12].Unit_code := 41, Detailed.element_data[12].result_measurement := 0.021727756, Detailed.element_data[13].Variable_code := 216, Detailed.element_data[13].prec_code := 3, Detailed.element_data[13].Unit_code := 41, Detailed.element_data[13].result_measurement := 0.00085681677, Detailed.element_data[14].Variable_code := 218, Detailed.element_data[14].prec_code := 3, Detailed.element_data[14].Unit_code := 41, Detailed.element_data[14].result_measurement := 0.01094304, Detailed.element_data[15].Variable_code := 295, Detailed.element_data[15].prec_code := 3, Detailed.element_data[15].Unit_code := 12, Detailed.element_data[15].result_measurement := 5.0711865);
   CurrentDUTData : udt_DUTHistory[2] := ([0].Barcode := '260382826C', [0].VolumeTest := 159.86131, [0].LeakTest := -0.051409006, [1].Barcode := '260911463C', [1].VolumeTest := 191.42384, [1].LeakTest := 0.10728836);
   DryCycle_N1Ready : BOOL;
   DryCycle_N2Ready : BOOL;
   DUTHistoryDump : udt_DUTHistory := (Barcode := '260360509C', VolumeTest := 163.52058, LeakTest := -999.0);
   DUTTestHistory : udt_DUTHistory[10] := ([0].Barcode := '260291637C', [0].VolumeTest := 156.89374, [0].LeakTest := 0.12293458, [1].Barcode := '260380809C', [1].VolumeTest := 156.82765, [1].LeakTest := 0.13411045, [2].Barcode := '260281530C', [2].VolumeTest := 156.6537, [2].LeakTest := 0.12908131, [3].Barcode := '260382497C', [3].VolumeTest := 156.76877, [3].LeakTest := 0.11958182, [4].Barcode := '261530405C', [4].VolumeTest := 154.13881, [4].LeakTest := 0.10728836, [5].Barcode := '261520175C', [5].VolumeTest := 157.14537, [5].LeakTest := 0.10281801, [6].Barcode := '260911450C', [6].VolumeTest := 156.1754, [6].LeakTest := 0.11622906, [7].Barcode := '260382826C', [7].VolumeTest := 156.68964, [7].LeakTest := 0.11678785, [8].Barcode := '260350215C', [8].VolumeTest := 156.9294, [8].LeakTest := 0.11175871, [9].Barcode := '260911463C', [9].VolumeTest := 191.42384, [9].LeakTest := 0.10728836);
   EIPTemplateCommStatus : AOI_CommStatus;
   EIPTemplateDeviceInput : udt_EIPTemplateData;
   EIPTemplateDeviceOutput : udt_EIPTemplateData;
   EIPTemplateLocalInput : udt_EIPTemplateLocalInput;
   EIPTemplateLocalOutput : udt_EIPTemplateLocalOutput;
   FailCount : COUNTER := (PRE := 10);
   FaultsAndWarnings : STRING[96] := ([0] := 'Main power off', [1] := 'Main air not OK', [2] := 'EStop high', [3] := 'Guard doors open', [4] := 'Reject bin missing', [5] := 'No EIP connection to barcode scanner', [6] := 'No EIP connection to CTS1', [7] := 'No EIP connection to CTS2', [8] := 'No EIP connection to Robot', [9] := 'EStop Safety Block faulted', [10] := 'Barcode scanner fault', [11] := 'CTS1 fault', [12] := 'CTS2 fault', [13] := 'Robot fault', [14] := 'Robot gripper in unknown state', [15] := 'Conveyor alarm high', [16] := 'Cylinder 1 fault', [17] := 'Cylinder 2 fault', [18] := '24V DC not OK', [19] := 'Check conveyor cleat sensor', [32] := '3 in a row fault', [33] := '5 in an hour fault', [34] := '10 in a shift fault', [42] := 'Homing cycle overtime', [43] := 'Fail chute failed to register unit (Homing Seq)', [44] := 'Fail chute failed to register unit (Auto Seq)', [45] := 'Cylinder 1 down timeout', [46] := 'Cylinder 2 down timeout', [47] := 'Cylinder 1 up timeout', [48] := 'Cylinder 2 up timeout', [49] := 'Cylinder 1 movement requested but RFID not matching expected value.', [50] := 'Cylinder 2 movement requested but RFID not matching expected value.', [64] := 'Cycle stop requested', [65] := 'Cycle pause requested', [66] := 'Step mode active', [67] := 'Dry cycle active', [68] := 'MES bypass active', [74] := 'Main sequence stuck on step$0D$0A', [75] := 'Homing sequence stuck on step$0D$0A', [76] := 'CTS1 sequence stuck on step 9000', [77] := 'CTS2 sequence stuck on step 9000', [78] := 'Conveyor sequence stuck on step 0', [79] := 'Main sequence stuck on step$0D$0A', [80] := 'Homing sequence stuck on step$0D$0A', [81] := 'CTS1 sequence stuck on step ', [82] := 'CTS2 sequence stuck on step ', [83] := 'Conveyor sequence stuck on step ', [84] := 'CTS1 test requested but interlock not met', [85] := 'CTS2 test requested but interlock not met', [86] := 'CTS1 not ready', [87] := 'CTS2 not ready', [88] := 'Robot movement requested but interlock not met', [89] := 'Conveyor movement requested but interlock not met', [90] := 'Nest 1 movement requested but interlock not met', [91] := 'Nest 2 movement requested but interlock not met', [94] := 'Fail bin full, please empty');
   FFLU_CTS1Leak : CONTROL := (LEN := 10, POS := 10, DN := 1);
   FFLU_CTS1Vol : CONTROL := (LEN := 10, POS := 10, DN := 1);
   FFLU_CTS2Leak : CONTROL := (LEN := 10, POS := 10, DN := 1);
   FFLU_CTS2Vol : CONTROL := (LEN := 10, POS := 10, DN := 1);
   FFLU_DUTHistory : CONTROL := (LEN := 10, POS := 10, DN := 1);
   FFLUDumpREAL : REAL;
   HMI_CloseDisplay : DINT := 12;
   HMI_OP220_ClearProcessFaultCounts_IND : BOOL;
   HMI_OP220_ClearProcessFaultCounts_PB : BOOL;
   HMI_TestPointer : DINT;
   HomingClearNestsBypass : BOOL := 1;
   InfeedCounter : COUNTER := (PRE := 9999999, ACC := 50);
   LastFaults : DINT[2] := ([0] := 1057263);
   LastShiftNumber : DINT := 2;
   LeakTester1 : udt_OutputStructure := (REQ := 3);
   LeakTester2 : udt_OutputStructure := (REQ := 3);
   Mode_CapActuators : BOOL;
   Mode_CapCTS : BOOL;
   Mode_CapCylinders : BOOL;
   Mode_CapFail : BOOL;
   Mode_CapPass : BOOL;
   Mode_CapRobot : BOOL;
   Mode_CapShuffle : BOOL;
   Nest1Bypass : BOOL := 1;
   Nest1Cylinder : udt_OutputStructure := (IL := 1, BTMR.PRE := 500);
   Nest1Empty : BOOL;
   Nest1Ready : BOOL;
   Nest2Bypass : BOOL;
   Nest2Cylinder : udt_OutputStructure := (IL := 1, BTMR.PRE := 500);
   Nest2Empty : BOOL := 1;
   Nest2Ready : BOOL;
   ONS_AutoMode : BOOL := 1;
   ONS_CapActuators : BOOL;
   ONS_CapCTS : BOOL;
   ONS_CapCylinders : BOOL;
   ONS_CapFail : BOOL;
   ONS_CapPass : BOOL;
   ONS_CapRobot : BOOL;
   ONS_CapShuffle : BOOL;
   ONS_ClearWarnings : BOOL;
   ONS_CTS1ClearResultsBC : BOOL := 1;
   ONS_CTS1GetResults : BOOL;
   ONS_CTS1ResultHistory : BOOL;
   ONS_CTS2ClearResultsBC : BOOL := 1;
   ONS_CTS2GetResults : BOOL;
   ONS_CTS2ResultHistory : BOOL;
   ONS_CycleStop : BOOL;
   ONS_FailBinRemoved : BOOL;
   ONS_HMICloseDisplay : BOOL := 1;
   ONS_ManuMode : BOOL := 1;
   ONS_RobotGripper : SINT := 1;
   OP220 : udt_Mode := (PowerOn := 1, PowerOnONS := 1, AirOk := 1, UtilitiesOk := 1, EStopsOk := 1, GuardDoorsOk := 1, FaultActive := 1, WarningActive := 1, ReadyForAuto := 1, ManualMode := 1, StepModeToggle := 1, Home := 1, MESBypass := 1, ManualMode_IND := 2, Home_IND := 2, HMIBackgroundIND := 2, Faults[0] := 1057263, Warnings[0] := 16, HomingOvertime.PRE := 120000, PowerOnTMR.PRE := 500, PowerOnTMR.ACC := 500, PowerOnTMR.EN := 1, PowerOnTMR.DN := 1, AirOKTMR.PRE := 500, AirOKTMR.ACC := 500, AirOKTMR.EN := 1, AirOKTMR.DN := 1, CycleStopOverideTMR.PRE := 3000, FaultTMR[0].TMR[0].PRE := 1, FaultTMR[0].TMR[1].PRE := 1, FaultTMR[0].TMR[2].PRE := 1, FaultTMR[0].TMR[3].PRE := 1, FaultTMR[0].TMR[4].PRE := 60000, FaultTMR[0].TMR[5].PRE := 1000, FaultTMR[0].TMR[6].PRE := 1000, FaultTMR[0].TMR[7].PRE := 1000, FaultTMR[0].TMR[8].PRE := 1000, FaultTMR[0].TMR[9].PRE := 1, FaultTMR[0].TMR[10].PRE := 1, FaultTMR[0].TMR[11].PRE := 1, FaultTMR[0].TMR[12].PRE := 1, FaultTMR[0].TMR[13].PRE := 1, FaultTMR[0].TMR[14].PRE := 1, FaultTMR[0].TMR[15].PRE := 1000, FaultTMR[0].TMR[16].PRE := 1, FaultTMR[0].TMR[17].PRE := 1, FaultTMR[0].TMR[18].PRE := 1, FaultTMR[0].TMR[19].PRE := 1, FaultTMR[1].TMR[0].PRE := 1, FaultTMR[1].TMR[1].PRE := 1, FaultTMR[1].TMR[2].PRE := 1, FaultTMR[1].TMR[10].PRE := 1, FaultTMR[1].TMR[11].PRE := 1, FaultTMR[1].TMR[12].PRE := 1, FaultTMR[1].TMR[13].PRE := 1, FaultTMR[1].TMR[14].PRE := 1, FaultTMR[1].TMR[15].PRE := 1, FaultTMR[1].TMR[16].PRE := 1, FaultTMR[1].TMR[17].PRE := 1, FaultTMR[1].TMR[18].PRE := 1,
        FaultTMR[1].TMR[19].PRE := 1, FaultTMR[1].TMR[20].PRE := 1, WarningTMR[0].TMR[0].PRE := 1, WarningTMR[0].TMR[1].PRE := 1, WarningTMR[0].TMR[2].PRE := 1, WarningTMR[0].TMR[3].PRE := 1, WarningTMR[0].TMR[4].PRE := 1, WarningTMR[0].TMR[4].ACC := 1, WarningTMR[0].TMR[4].EN := 1, WarningTMR[0].TMR[4].DN := 1, WarningTMR[0].TMR[10].PRE := 1, WarningTMR[0].TMR[11].PRE := 1, WarningTMR[0].TMR[12].PRE := 1, WarningTMR[0].TMR[13].PRE := 1, WarningTMR[0].TMR[14].PRE := 1, WarningTMR[0].TMR[20].PRE := 2000, WarningTMR[0].TMR[21].PRE := 2000, WarningTMR[0].TMR[22].PRE := 30000, WarningTMR[0].TMR[23].PRE := 30000, WarningTMR[0].TMR[24].PRE := 5000, WarningTMR[0].TMR[25].PRE := 1000, WarningTMR[0].TMR[26].PRE := 1000, WarningTMR[0].TMR[27].PRE := 1000, WarningTMR[0].TMR[30].PRE := 1);
   OP220_Disable3510 : BOOL;
   OP220_Fault_Counter : COUNTER := (PRE := 9999999, ACC := 200);
   OP220_Fault_Counter_ONS : BOOL;
   OP220_Fault_Number : DINT;
   OP220_Fault_Reset_ONS : BOOL;
   OP220_FaultCounter_Reset_ONS : BOOL;
   OP220_HomeONS : BOOL;
   OP220_HomingSeq : udt_SequenceStructure_X64 := (SequenceRunning := 1, CurrentStep := 1160, NextStep := 1170, StepHistory[0] := 1000, StepHistory[1] := 1020, StepHistory[2] := 1030, StepHistory[3] := 1120, StepHistory[4] := 1140, StepHistory[5] := 1160, StepHistory[6] := 9000, StepHistory[7] := 1000, StepHistory[8] := 1020, StepHistory[9] := 1030, StepHistory[10] := 1120, StepHistory[11] := 1140, StepHistory[12] := 1160, StepHistory[13] := 9000, StepHistory[14] := 1000, StepHistory[15] := 1020, StepHistory[16] := 1030, StepHistory[17] := 1120, StepHistory[18] := 1140, StepHistory[19] := 1160, StepHistory[20] := 1180, StepHistory[21] := 1000, StepHistory[22] := 1020, StepHistory[23] := 1030, StepHistory[24] := 1140, StepHistory[25] := 1160, StepHistory[26] := 1180, StepHistory[27] := 1000, StepHistory[28] := 1020, StepHistory[29] := 1030, StepHistory[30] := 1140, StepHistory[31] := 1160, StepHistory[32] := 1180, StepHistory[33] := 1000, StepHistory[34] := 1020, StepHistory[35] := 1030, StepHistory[36] := 1140, StepHistory[37] := 1160, StepHistory[38] := 1180, StepHistory[39] := 1000, StepHistory[40] := 1020, StepHistory[41] := 1030, StepHistory[42] := 1140, StepHistory[43] := 1160, StepHistory[44] := 1180, StepHistory[45] := 1000, StepHistory[46] := 1020, StepHistory[47] := 1030, StepHistory[48] := 1140, StepHistory[49] := 1160, StepHistory[50] := 1180, StepHistory[51] := 1000, StepHistory[52] := 1020, StepHistory[53] := 1030, StepHistory[54] := 1120, StepHistory[55] := 1140, StepHistory[56] := 1160,
        StepHistory[57] := 1180, StepHistory[58] := 1000, StepHistory[59] := 1020, StepHistory[60] := 1030, StepHistory[61] := 1120, StepHistory[62] := 1140, StepHistory[63] := 1160, StepDescriptionPointer := 1, CurrentCycleTime := 139.077, AverageCycleTime := 0.0184, PreviousCycleTime := 3374.766, CycleTimeHistory[0] := 0.004, CycleTimeHistory[1] := 0.057, CycleTimeHistory[3] := 0.048, CycleTimeHistory[5] := 0.043, CycleTimeHistory[7] := 0.032, CurrentStepCycleTime := 1016.759, StepTimeHistory[3] := 0.038, StepTimeHistory[4] := 0.038, StepTimeHistory[5] := 0.038, StepTimeHistory[10] := 0.028, StepTimeHistory[11] := 0.028, StepTimeHistory[12] := 0.028, StepTimeHistory[20] := 2203.91, StepTimeHistory[21] := 2203.91, StepTimeHistory[22] := 2203.91, StepTimeHistory[23] := 2203.91, StepTimeHistory[24] := 2203.91, StepTimeHistory[25] := 2203.91, StepTimeHistory[26] := 727.29, StepTimeHistory[27] := 727.29, StepTimeHistory[28] := 727.29, StepTimeHistory[29] := 727.29, StepTimeHistory[30] := 727.29, StepTimeHistory[31] := 727.29, StepTimeHistory[32] := 1442.421, StepTimeHistory[33] := 1442.421, StepTimeHistory[34] := 1442.421, StepTimeHistory[35] := 1442.421, StepTimeHistory[36] := 1442.421, StepTimeHistory[37] := 1442.421, StepTimeHistory[38] := 1.302, StepTimeHistory[39] := 1.302, StepTimeHistory[40] := 1.302, StepTimeHistory[41] := 1.302, StepTimeHistory[42] := 1.302, StepTimeHistory[43] := 1.302, StepTimeHistory[44] := 18.821, StepTimeHistory[45] := 18.821, StepTimeHistory[46] := 18.821, StepTimeHistory[47] := 18.821, StepTimeHistory[48] := 18.821, StepTimeHistory[49] := 18.821, StepTimeHistory[50] := 1539.229, StepTimeHistory[51] := 1539.229, StepTimeHistory[52] := 1539.229, StepTimeHistory[53] := 1539.229, StepTimeHistory[54] := 0.05, StepTimeHistory[55] := 0.05, StepTimeHistory[56] := 0.05,
        StepTimeHistory[57] := 372.918, StepTimeHistory[58] := 372.918, StepTimeHistory[59] := 372.918, StepTimeHistory[60] := 372.918, StepTimeHistory[61] := 0.05, StepTimeHistory[62] := 0.05, StepTimeHistory[63] := 0.05, StepTimer.PRE := 999999999, CycleTimer.PRE := 999999999, CycleTimer.ACC := 139079, CycleTimer.EN := 1, CycleTimer.TT := 1);
   OP220_LeakTest : udt_ProcessFault := (ShiftCount := 3);
   OP220_PartToPartCycleTMR : TIMER := (PRE := 999999999);
   OP220_ProcessFaultsONS : DINT;
   OP220_Seq : udt_SequenceStructure_X64 := (ONS := 2, StepHistory[0] := 2530, StepHistory[1] := 2540, StepHistory[2] := 2550, StepHistory[4] := 1000, StepHistory[5] := 2500, StepHistory[6] := 2510, StepHistory[8] := 1000, StepHistory[9] := 2500, StepHistory[10] := 2510, StepHistory[11] := 2520, StepHistory[12] := 2530, StepHistory[13] := 2540, StepHistory[14] := 2550, StepHistory[15] := 2560, StepHistory[16] := 2570, StepHistory[17] := 2580, StepHistory[18] := 9000, StepHistory[19] := 1000, StepHistory[20] := 3500, StepHistory[21] := 3510, StepHistory[22] := 3520, StepHistory[23] := 3530, StepHistory[24] := 3540, StepHistory[25] := 3550, StepHistory[26] := 9000, StepHistory[27] := 1000, StepHistory[28] := 2500, StepHistory[29] := 2510, StepHistory[30] := 2520, StepHistory[31] := 2530, StepHistory[32] := 2540, StepHistory[33] := 2550, StepHistory[34] := 2560, StepHistory[35] := 2570, StepHistory[36] := 2580, StepHistory[37] := 9000, StepHistory[38] := 1000, StepHistory[39] := 3500, StepHistory[40] := 3510, StepHistory[41] := 3520, StepHistory[42] := 3530, StepHistory[43] := 3540, StepHistory[44] := 3550, StepHistory[45] := 9000, StepHistory[46] := 1000, StepHistory[47] := 2500, StepHistory[48] := 2510, StepHistory[49] := 2520, StepHistory[50] := 2530, StepHistory[51] := 2540, StepHistory[52] := 2550, StepHistory[53] := 2560, StepHistory[54] := 2570, StepHistory[55] := 2580, StepHistory[56] := 9000, StepHistory[57] := 1000, StepHistory[58] := 3500, StepHistory[59] := 3510, StepHistory[60] := 3520,
        StepHistory[61] := 3530, StepHistory[62] := 3540, StepHistory[63] := 3550, StepDescriptionPointer := 1, AverageCycleTime := 41.43, PreviousCycleTime := 5.431, CycleTimeHistory[0] := 15.582, CycleTimeHistory[1] := 266.467, CycleTimeHistory[2] := 15.644, CycleTimeHistory[3] := 15.211, CycleTimeHistory[4] := 15.596, CycleTimeHistory[5] := 5.52, CycleTimeHistory[6] := 43.678, CycleTimeHistory[7] := 5.365, CycleTimeHistory[8] := 25.806, CycleTimeHistory[9] := 5.431, CurrentStepCycleTime := 446.276, StepTimeHistory[0] := 0.679, StepTimeHistory[1] := 0.059, StepTimeHistory[2] := 0.541, StepTimeHistory[3] := 0.541, StepTimeHistory[4] := 0.541, StepTimeHistory[5] := 0.029, StepTimeHistory[6] := 16.795, StepTimeHistory[7] := 16.795, StepTimeHistory[8] := 16.795, StepTimeHistory[9] := 0.061, StepTimeHistory[10] := 0.709, StepTimeHistory[11] := 0.059, StepTimeHistory[12] := 0.673, StepTimeHistory[13] := 0.065, StepTimeHistory[14] := 1.229, StepTimeHistory[15] := 0.139, StepTimeHistory[16] := 2.044, StepTimeHistory[17] := 0.53, StepTimeHistory[18] := 0.53, StepTimeHistory[19] := 12.272, StepTimeHistory[20] := 0.068, StepTimeHistory[21] := 1.239, StepTimeHistory[22] := 0.079, StepTimeHistory[23] := 0.749, StepTimeHistory[24] := 0.069, StepTimeHistory[25] := 29.196, StepTimeHistory[26] := 29.196, StepTimeHistory[27] := 29.196, StepTimeHistory[28] := 0.06, StepTimeHistory[29] := 0.699, StepTimeHistory[30] := 0.069, StepTimeHistory[31] := 0.675, StepTimeHistory[32] := 0.062, StepTimeHistory[33] := 1.22, StepTimeHistory[34] := 0.069, StepTimeHistory[35] := 1.979, StepTimeHistory[36] := 0.522, StepTimeHistory[37] := 0.522, StepTimeHistory[38] := 12.265, StepTimeHistory[39] := 0.079, StepTimeHistory[40] := 1.209, StepTimeHistory[41] := 0.069, StepTimeHistory[42] := 0.779,
        StepTimeHistory[43] := 0.069, StepTimeHistory[44] := 11.329, StepTimeHistory[45] := 11.329, StepTimeHistory[46] := 11.329, StepTimeHistory[47] := 0.067, StepTimeHistory[48] := 0.699, StepTimeHistory[49] := 0.069, StepTimeHistory[50] := 0.677, StepTimeHistory[51] := 0.061, StepTimeHistory[52] := 1.229, StepTimeHistory[53] := 0.089, StepTimeHistory[54] := 1.984, StepTimeHistory[55] := 0.546, StepTimeHistory[56] := 0.546, StepTimeHistory[57] := 12.28, StepTimeHistory[58] := 0.075, StepTimeHistory[59] := 1.219, StepTimeHistory[60] := 0.059, StepTimeHistory[61] := 0.769, StepTimeHistory[62] := 0.059, StepTimeHistory[63] := 446.276, StepTimer.PRE := 999999999, CycleTimer.PRE := 999999999);
   OutfeedCounter : COUNTER := (PRE := 9999999, ACC := 26217);
   ResetFeedCounters : BOOL;
   RFID_CmdNest1 : BOOL;
   RFID_CmdNest2 : BOOL;
   RFID_Comp : AOI_RFIDCompare;
   RFID_Cylinder1_Mismatch : BOOL;
   RFID_Cylinder2_Mismatch : BOOL;
   RFID_DiagData : DINT[4];
   RFID_DoneONS : BOOL;
   RFID_EntryStatus : DINT;
   RFID_ExpectedFixtureVal : SINT[5,12] := ([1,0] := 26, [1,1] := 6, [1,2] := 2, [1,3] := 26, [1,5] := 7, [1,6] := 4, [1,7] := 1, [1,8] := 3, [1,10] := 1, [1,11] := 1, [2,0] := 50, [2,1] := 54, [2,2] := 48, [2,3] := 54, [2,4] := 48, [2,5] := 50, [2,6] := 50, [2,7] := 54, [2,8] := 48, [2,9] := 48, [2,10] := 48, [2,11] := 55, [3,0] := 48, [3,1] := 52, [3,2] := 48, [3,3] := 48, [3,4] := 48, [3,5] := 48, [3,6] := 48, [3,7] := 48, [3,8] := 48, [3,9] := 48, [3,10] := 48, [3,11] := 48);
   RFID_FSC : TIMER;
   RFID_HMI_ExecuteRequest : BOOL;
   RFID_LoadingNestDiagData : DINT[4];
   RFID_LoadingNestReceiveBuffer : SINT[8000];
   RFID_LoadingNestSendBuffer : SINT[8000];
   RFID_Mismatch : BOOL;
   RFID_Nest2Delay : TIMER := (PRE := 200);
   RFID_NewRead : BOOL;
   RFID_PortOffset : DINT;
   RFID_ReadData : STR_RFID := 'LUFFY$00$00$00$00$00$00$00$00$00$00$00$00$00$00$00$00$00$00$00';
   RFID_ReceiveBuffer : SINT[8000];
   RFID_RWHAllPort : RWH_CMD := (ixConnOK := 1, isiModuleID := 13, isiFunctionID := 4, iiRdWrLength := 40, odiStatus := 16#0000_7000, oxTagPresent := 1);
   RFID_Search_Ctrl : CONTROL := (LEN := 40, POS := 5, EN := 1, IN := 1, FD := 1);
   RFID_SendBuffer : SINT[8000];
   RFID_TagStatus : BOOL[32] := ([1] := 1, [3] := 1);
   RFIDBypass : BOOL;
   RFIDLoadingNestScanner : udt_OutputStructure;
   RFIDScanner : udt_OutputStructure := (IL := 1, REQ := 1);
   Robot : udt_OutputStructure := (IL := 1, BC := 1, REQ := 1);
   RobotGripper : udt_OutputStructure := (IL := 1, BTMR.PRE := 2000);
   RobotInputs : udt_EpsonInputs := (ib_Ready := 1, ib_MotorsOn := 1, ib_IsHome := 1, ib_InPos := 1, ib_GripOpen := 1, iW_PositionEcho := 1, iR_X := 189.53908, iR_Y := 109.599014, iR_Z := -56.044655, iR_U := -217.60461);
   RobotOutputs : udt_EpsonOutputs := (ob_SpeedOverride := 1, oB_SpeedPerc := 100, oW_TargetPosition := 1, oR_X := 191.0, oR_Y := -84.0, oR_Z := -52.0, oR_U := -270.0);
   ShiftTimes : SINT[24] := ([0] := 7, [1] := 15, [2] := 23, [3] := -1, [4] := -1, [5] := -1, [6] := -1, [7] := -1, [8] := -1, [9] := -1, [10] := -1, [11] := -1, [12] := -1, [13] := -1, [14] := -1, [15] := -1, [16] := -1, [17] := -1, [18] := -1, [19] := -1, [20] := -1, [21] := -1, [22] := -1, [23] := -1);
   TempConsumedFromPLC : BOOL;
   TempStrBuff : STRING[10] := ([0] := '0', [1] := '/', [2] := '0', [3] := ')');
   TON_CapActuatorsDelay : TIMER := (PRE := 5000);
   TON_CapActuatorsDelay2 : TIMER := (PRE := 100);
   TON_CapCTSDelay : TIMER := (PRE := 2000);
   TON_CapCTSDelay2 : TIMER := (PRE := 2000);
   TON_CapCylindersDelay : TIMER := (PRE := 5500);
   TON_CapShuffleCTS1Delay : TIMER := (PRE := 5000);
   TON_CapShuffleCTS2Delay : TIMER := (PRE := 5000);
   TON_ConveyorCleatTimeout : TIMER := (PRE := 5000);
   TON_ConvUnloadDelay : TIMER := (PRE := 300);
   TON_CTS1GetResultRetry : TIMER := (PRE := 1000);
   TON_CTS1GetResultTimeout : TIMER := (PRE := 1000);
   TON_CTS1NotGettingResultsTimeout : TIMER := (PRE := 1000);
   TON_CTS1Trigger0 : TIMER := (PRE := 200);
   TON_CTS1Trigger1 : TIMER := (PRE := 200);
   TON_CTS1Trigger2 : TIMER := (PRE := 200);
   TON_CTS2GetResultRetry : TIMER := (PRE := 1000);
   TON_CTS2GetResultTimeout : TIMER := (PRE := 1000);
   TON_CTS2NotGettingResultsTimeout : TIMER := (PRE := 1000);
   TON_CTS2Trigger0 : TIMER := (PRE := 200);
   TON_CTS2Trigger1 : TIMER := (PRE := 200);
   TON_CTS2Trigger2 : TIMER := (PRE := 1000);
   TON_Cylinder1DownTimeout : TIMER := (PRE := 5000);
   TON_Cylinder1UpTimeout : TIMER := (PRE := 5000);
   TON_Cylinder2DownTimeout : TIMER := (PRE := 5000);
   TON_Cylinder2UpTimeout : TIMER := (PRE := 5000);
   TON_FailChute : TIMER[10] := ([0].PRE := 1000, [1].PRE := 1000, [2].PRE := 1000, [3].PRE := 1000);
   TON_HMICloseDisplayDelay : TIMER := (PRE := 500);
   TON_Nest1CylinderTimer : TIMER := (PRE := 5000);
   TON_Nest1DryCycleDryTest : TIMER := (PRE := 5000);
   TON_Nest2CylinderTimer : TIMER := (PRE := 5000);
   TON_Nest2DryCycleDryTest : TIMER := (PRE := 5000);
   TON_RobotPickupSafeDelay : TIMER := (PRE := 200, ACC := 500, EN := 1, DN := 1);
   TON_RobotReqRetry : TIMER := (PRE := 1000);
   TON_RobotReqTimeout : TIMER := (PRE := 1000);
END_VAR
